// TIA Portal V16 export
// export: Created 2021-09-08T12:46:15.9434671Z, ExportSetting WithDefaults, DisplayName Totally Integrated Automation Portal, DisplayVersion V16 Update 3, DisplayName TIA Portal Version Control Interface, DisplayVersion V16 Update 2, DisplayName TIA Portal Openness, DisplayVersion V16 Update 3, DisplayName TIA Portal Teamcenter Gateway, DisplayVersion V16, DisplayName STEP 7 Professional, DisplayVersion V16 Update 3, DisplayName STEP 7 Safety, DisplayVersion V16, DisplayName WinCC Advanced, DisplayVersion V16 Update 3
TYPE "UZ_Data"
// stored: IsFailsafeCompliant false
   STRUCT
      Ready { ExternalAccessible := 'False'; ExternalVisible := 'False'; ExternalWritable := 'False'} : Bool;   // Drive ready to start
      Fault { ExternalAccessible := 'False'; ExternalVisible := 'False'; ExternalWritable := 'False'} : Bool;   // Fault is present. Trip or Trip lock
      Warning { ExternalAccessible := 'False'; ExternalVisible := 'False'; ExternalWritable := 'False'} : Bool;   // Warning present
      Running : Bool;   // Drive is started but not necessarily running on reference speed.
      Run_On_ref { ExternalAccessible := 'False'; ExternalVisible := 'False'; ExternalWritable := 'False'} : Bool;   // Running on reference
      MotorCurrent : Real;   // Actual motor Current
      MotorPower : Real;   // Motor Power
      MAV : Real;   // Main Actual Value read from Drive 0 - 100.00%
      comErr { ExternalAccessible := 'False'; ExternalVisible := 'False'; ExternalWritable := 'False'} : Int;   // Result of DPRD_DAT 0=No error
      ErrorConnection : Bool;   // Present Error DPRD_DAT
   END_STRUCT;
END_TYPE
